(* IEC 61131-3 sources: lc3-lib/Button, 3 files *)

(* ---- Toggle.iecfbd ---- *)
FUNCTION Toggle
  VAR_INPUT
    in : BOOL;
    value : BOOL;
  END_VAR
  VAR_OUTPUT
    out : BOOL;
  END_VAR

  (*

    // Network 1:
    NOT(IN := value, NOT => @C(7).NOT);
    SEL(G := in, IN0 := value, IN1 := @C(7).NOT, SEL => out);

  *)

  @C(1) : @F(SEL), @R(530.0, 260.0, 120.0, 58.0), BOOL, @I(@N(G), @L(9.5)), @I(@N(IN0), @L(29.5)), @I(@N(IN1), @L(49.5)), @O(@N(SEL), @R(9.5));
  @VF(2) : @E(in), @R(300.0, 260.0, 140.0, 19.0);
  @VF(4) : @E(value), @R(300.0, 280.0, 140.0, 19.0);
  @VF(5) : @E(out), @R(700.0, 260.0, 140.0, 19.0);
  @C(7) : @F(NOT), @R(450.0, 300.0, 60.0, 18.5), BOOL, @I(@N(IN), @L(9.5)), @O(@N(NOT), @R(9.5));
  @VF(10) : @E(value), @R(300.0, 300.0, 140.0, 19.0);

  @G(3) :
     @L(@VF(2).o, @C(1).G)
    ;
  @G(6) :
     @L(@C(1).SEL, @VF(5).i)
    ;
  @G(8) :
     @L(@C(7).NOT, @C(1).IN1)
    ;
  @G(9) :
     @L(@VF(4).o, @C(1).IN0)
    ;
  @G(11) :
     @L(@VF(10).o, @C(7).IN)
    ;
END_FUNCTION

(* ---- Multi_Click.iecfbd ---- *)
FUNCTION_BLOCK Multi_Click
  {
    height := 130;
  }

  VAR
    CTU1 : CTU;
    TOF1 : TOF;
    R_TRIG1 : R_TRIG;
    F_TRIG1 : F_TRIG;
  END_VAR
  VAR_INPUT
    in : BOOL;
    period : TIME := T#500ms;
    CV : INT;
  END_VAR
  VAR_OUTPUT
    out : BOOL;
  END_VAR

  (*

    // Network 1:
    TOF1(IN := in, PT := period);
    F_TRIG1(CLK := TOF1.Q);
    R_TRIG1(CLK := CTU1.Q);
    out := R_TRIG1.Q;
    OR(IN1 := F_TRIG1.Q, IN2 := R_TRIG1.Q, OR => @C(17).OR);
    CTU1(CU := in, R := @C(17).OR, PV := CV);

  *)

  @C(4) : @FB(CTU1), @R(930.0, 190.0, 100.0, 58.0), @I(@N(CU), @L(9.5)), @I(@N(R), @L(29.5)), @I(@N(PV), @L(49.5)), @O(@N(Q), @R(9.5)), @O(@N(CV), @R(49.5));
  @VF(9) : @E(in), @R(270.0, 180.0, 140.0, 19.0);
  @VF(10) : @E(out), @R(1300.0, 190.0, 140.0, 19.0);
  @C(5) : @FB(TOF1), @R(720.0, 40.0, 100.0, 38.0), @I(@N(IN), @L(9.5)), @I(@N(PT), @L(29.5)), @O(@N(Q), @R(9.5)), @O(@N(ET), @R(29.5));
  @VF(6) : @E(period), @R(530.0, 60.0, 140.0, 19.0);
  @OLT(12) : @R(1110.0, 240.0, 80.0, 18.0), @S(@C(4).CV);
  @OLT(13) : @R(360.0, 110.0, 80.0, 18.0), @S(@VF(9).o);
  @C(1) : @FB(R_TRIG1), @R(1069.9, 193.0, 140.0, 18.5), @I(@N(CLK), @L(9.5)), @O(@N(Q), @R(9.5));
  @C(14) : @FB(F_TRIG1), @R(600.0, 130.0, 140.0, 18.5), @I(@N(CLK), @L(9.5)), @O(@N(Q), @R(9.5));
  @C(17) : @F(OR), @R(800.0, 130.0, 40.0, 38.0), BOOL, @I(@N(IN1), @L(9.5)), @I(@N(IN2), @L(29.5)), @O(@N(OR), @R(9.5));
  @VF(2) : @E(CV), @R(270.0, 230.0, 140.0, 19.0);
  @CP(11) : 497.0, 189.5;
  @CP(21) : 1236.0, 193.5;

  @G(3) :
     @L(@VF(9).o, @CP(11)),
     @L(@CP(11), @C(4).CU),
     @L(@CP(11), @C(5).IN)
    ;
  @G(7) :
     @L(@VF(6).o, @C(5).PT)
    ;
  @G(15) :
     @L(@C(1).Q, @CP(21)),
     @L(@CP(21), @VF(10).i),
     @L(@CP(21), @C(17).IN2)
    ;
  @G(16) :
     @L(@C(4).Q, @C(1).CLK)
    ;
  @G(18) :
     @L(@C(5).Q, @C(14).CLK)
    ;
  @G(19) :
     @L(@C(14).Q, @C(17).IN1)
    ;
  @G(20) :
     @L(@C(17).OR, @C(4).R)
    ;
  @G(8) :
     @L(@VF(2).o, @C(4).PV)
    ;
END_FUNCTION_BLOCK

(* ---- Multi_Click.iecst ---- *)
FUNCTION_BLOCK Multi_Click
  {
    height := 150;
    width := 120;
  }
	VAR_INPUT
		in : BOOL;
		period : TIME := T#300ms;
	END_VAR
	VAR_OUTPUT
		out : BOOL;
		cv : UINT;
	END_VAR
	VAR
		trigger_in : R_TRIG;
		timer : TOF;
		trigger_timer : F_TRIG;
		cv_reset : BOOL;
	END_VAR

	IF trigger_timer.Q THEN
		cv := 0;
	END_IF;

	timer(IN := in, PT := period);

	trigger_in(CLK := in);
	IF trigger_in.Q THEN
		cv := cv + 1;
	END_IF;

	trigger_timer(CLK := timer.Q, Q => out);
END_FUNCTION_BLOCK

FUNCTION_BLOCK Double_Click
  {
    height := 120;
    width := 120;
  }
	VAR_INPUT
		in : BOOL;
		period : TIME := T#300ms;
	END_VAR
	VAR_OUTPUT
		out : BOOL;
	END_VAR
	VAR
		multi_click : Multi_Click;
	END_VAR
	multi_click(in := in, period := period);
	out := multi_click.out AND multi_click.cv = 2;
END_FUNCTION_BLOCK
